// TIA Portal V20 export
// export: Created 2026-04-11T06:02:30.2272393Z, ExportSetting WithDefaults, DisplayName Totally Integrated Automation Portal, DisplayVersion V20, DisplayName TIA Portal Openness, DisplayVersion V20, DisplayName TIA Portal Version Control Interface, DisplayVersion V20, DisplayName STEP 7 Professional, DisplayVersion V20, DisplayName STEP 7 Safety, DisplayVersion V20, DisplayName WinCC Basic/Comfort/Advanced, DisplayVersion V20, DisplayName WinCC Unified, DisplayVersion V20
TYPE "udtHMI_SiwarexCalibration"
// stored: IsFailsafeCompliant false
   STRUCT
      bPB_ZeroLoadCell : Bool;   // PB to zero the load cell
      bPBEN_ZeroLoadCell { ExternalWritable := 'False'} : Bool;   // Enable scale zeroing
      bPB_CalibrateWeight0 : Bool;   // PB to set current weight as calibration weight 0
      bPBEN_CalibrateWeight0 { ExternalWritable := 'False'} : Bool;   // Enable set calibration weight 0
      bPB_CalibrateWeight1 : Bool;   // PB to set current weight as calibration weight 1
      bPBEN_CalibrateWeight1 { ExternalWritable := 'False'} : Bool;   // Enable set calibration weight 1
      bPB_CalibrateWeight2 : Bool;   // PB to set current weight as calibration weight 2
      bPBEN_CalibrateWeight2 { ExternalWritable := 'False'} : Bool;   // Enable set calibration weight 2
      bPB_SetValues : Bool;   // PB to set calibration values
      bPBEN_SetValues { ExternalWritable := 'False'} : Bool;   // Enable setting of calibration values
      bPB_EnableCalibration : Bool;   // Toggles the enabling of calibration
      bTOG_EnableCalibration { ExternalWritable := 'False'} : Bool;   // Status of calibration enable
      bPB_ResetCalibration : Bool;   // PB to reset calibration routine
      bPB_ResetError : Bool;   // PB to reset error
      b3WeightCalibrationMode : Bool;   // Calibrates using 3 weights instead of 2
      bError { ExternalWritable := 'False'} : Bool;   // Error exists
      iModuleAddress : Int;   // IO address of module to calibrate
      iState { ExternalWritable := 'False'} : Int;   // State of the module calibration
      iErrorCode { ExternalWritable := 'False'} : Int;   // HMI error code
      iNumberOfDecimals { S7_SetPoint := 'True'} : Int;   // Number of decimals to display weight
      rCalibrationWeight0 { S7_SetPoint := 'True'} : Real;   // Value of calibration 0 weight
      rCalibrationWeight1 { S7_SetPoint := 'True'} : Real;   // Value of calibration 1 weight
      rCalibrationWeight2 { S7_SetPoint := 'True'} : Real;   // Value of calibration 2 weight
      rMaximumWeight { S7_SetPoint := 'True'} : Real;   // Maximum measurable weight
      rActualWeight { ExternalWritable := 'False'} : Real;   // Current weight measured by load cell
      rStandstillRange { S7_SetPoint := 'True'} : Real;   // Weight range of standstill
      rStandstillTime { S7_SetPoint := 'True'} : Real;   // Time needed to achieve standstill (s)
   END_STRUCT;
END_TYPE
